ABB RAPID module: TCP Server movement control v3.mod

MODULE TCP_MOVEMENT_CONTROL
    !2013-11-14

    !CONST jointtarget homePose:=[[0,0,0,0,0,0],[0,0,0,0,0,0]];
    CONST pos location:=[5000,-1000,1700];
    ![1758.41,-300,1752.13];
    CONST orient orientation:=[0.45,0.53,0.47,0.53];
    ![0.5471,-0.6908,0.1508,-0.448];
    CONST confdata configurationData:=[0,1,1,0];
    CONST extjoint externalJoints:=[4000,9E9,9E9,9E9,9E9,9E9];
    CONST robtarget homeTarget:=[location,orientation,configurationData,externalJoints];

    CONST byte msgOK{1}:=[1];
    CONST byte msgERR{1}:=[2];
    CONST byte msgDIS{1}:=[3];
    VAR byte msgVAR{1}:=[0];

    VAR pos currentPosition:=[0,0,0];

    VAR robtarget nextTarget:=[location,orientation,configurationData,externalJoints];

    VAR num stringToVal{3}:=[0,0,0];

        VAR num answer;
        VAR zonedata zone:=fine;

    ! Setup communication variables
    VAR socketdev temp_socket;
    VAR socketdev client_socket;
    VAR string received_string;
    VAR bool keep_listening:=TRUE;

    PROC parseStepAndMove()
        !VAR string str15 := "[600, 500, 225.3]";

        IF StrToVal(received_string,stringToVal) THEN
            !look at parsing
            TPWrite received_string+" Step parsed into "+NumToStr(stringToVal{1},0)+","+NumToStr(stringToVal{2},2)+","+NumToStr(stringToVal{3},0);
            !SocketSend client_socket\Data:=msgOK\NoOfBytes:=1;
        ELSE
            TPWrite "StrToVal("+received_string+") returned false";
            !SocketSend client_socket\Data:=msgERR\NoOfBytes:=1;
        ENDIF

        currentPosition:=CPos(\Tool:=tool0\WObj:=wobj0);

        IF currentPosition.x>5400 THEN
            msgVAR{1}:=1;
        ELSE
            msgVAR{1}:=0;
        ENDIF

        SocketSend client_socket\Data:=msgVAR\NoOfBytes:=1;

        msgVAR{1}:=0;

        !MoveL Offs(CRobT(\Tool:=tool0 \WObj:=wobj0), stringToVal{1} * stepSize, stringToVal{2} * stepSize, stringToVal{3} * stepSize),vmax,fine,tool0\WObj:=wobj0;
        MoveJ Offs(CRobT(\Tool:=tool0\WObj:=wobj0),stringToVal{1},stringToVal{2},stringToVal{3}),vmax,zone,tool0\WObj:=wobj0;
        stringToVal:=[0,0,0];
    ENDPROC

    PROC main()
        ConfL\Off;
        ConfJ\Off;

        !msgOK{1}:=[1];
        !msgERR{1}:=[2];
        !msgDIS{1}:=[3];

        !homeTarget:=[location,orientation,configurationData,externalJoints];
        MoveJ homeTarget,vmax,fine,tool0\WObj:=wobj0;

        TPReadFK answer,"Select Zone","fine","z50","z100","z150","z200";
        IF answer=1 THEN
            zone:=fine;
        ELSEIF answer=2 THEN
            zone:=z50;
        ELSEIF answer=3 THEN
            zone:=z100;
        ELSEIF answer=4 THEN
            zone:=z150;
        ELSEIF answer=5 THEN
            zone:=z200;
        ENDIF

        SocketCreate temp_socket;
        SocketBind temp_socket,"128.2.109.20",1025;
        SocketListen temp_socket;
        ! Waiting for a connection request
        SocketAccept temp_socket,client_socket;

        !Say OK to let the client know I'm alive
        SocketSend client_socket\Data:=msgOK\NoOfBytes:=1;

        WHILE keep_listening DO
            ! Communication
            SocketReceive client_socket\Str:=received_string;
            TPWrite "Client wrote: "+received_string;

            !Understand message
            IF received_string="Disconnect" THEN
                ! Shutdown the connection
                TPWrite "Shutdown acknowledged";
                keep_listening:=FALSE;
                !SocketSend client_socket\Data:=msgDIS\NoOfBytes:=1;
                !SocketSend client_socket\Str:="Shutdown acknowledged";
                SocketClose client_socket;
                !NEED TO BREAK OUT OF THE WHILE HERE
                !SocketSend socket1\Data:=msg_dc\NoOfBytes:=1;
            ELSE
                parseStepAndMove;
                !MoveJ parseStep(received_string),v20,z1,MyTool;
                !TPWrite "random debug statement";
            ENDIF

            received_string:="";
        ENDWHILE

        SocketClose temp_socket;
        TPWrite "Have a good one!";
    ENDPROC
ENDMODULE
